(* This function evaluates the Turbo ILK logic*)
(* The Turbo shall not Run if the vent valve is open*)
(* The function also switches off the Turbo if the Inlet pressure or the backing Pressure*)
(* are higher than the configured set point*)
FUNCTION F_TurboExtILKLogic : BOOL
VAR_INPUT
	Turbo		:	ST_PTM;
	BackingGauge:	ST_VG;
	InletGauge	:	ST_VG;
	VentValve	:	ST_VVC;
	ScrollPump	:	ST_RoughPump;
END_VAR

VAR
END_VAR

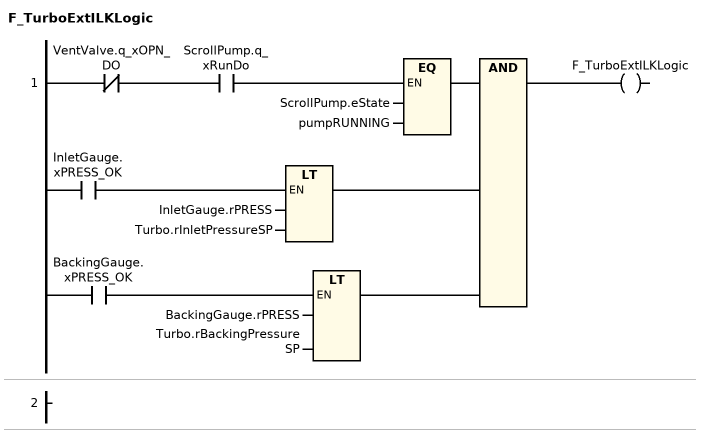
// NETWORK 1
F_TurboExtILKLogic := (NOT VentValve.q_xOPN_DO AND ScrollPump.q_xRunDo AND ScrollPump.eState = pumpRUNNING) AND (InletGauge.xPRESS_OK AND InletGauge.rPRESS < Turbo.rInletPressureSP) AND (BackingGauge.xPRESS_OK AND BackingGauge.rPRESS < Turbo.rBackingPressureSP);

// NETWORK 2

END_FUNCTION

(* stored: Version 1.1.0.1, ProductVersion 3.1.4022.18
   POU F_TurboExtILKLogic: Id {7245688f-5d30-4f2c-88b0-ff2e5b5ffecc}, SpecialFunc None *)
